ABB RobotStudio station: Mark3.rspag

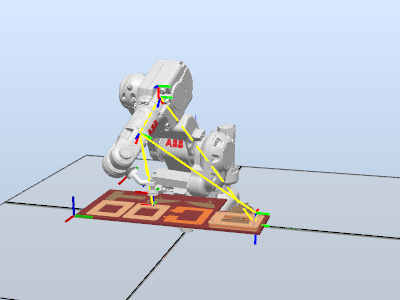
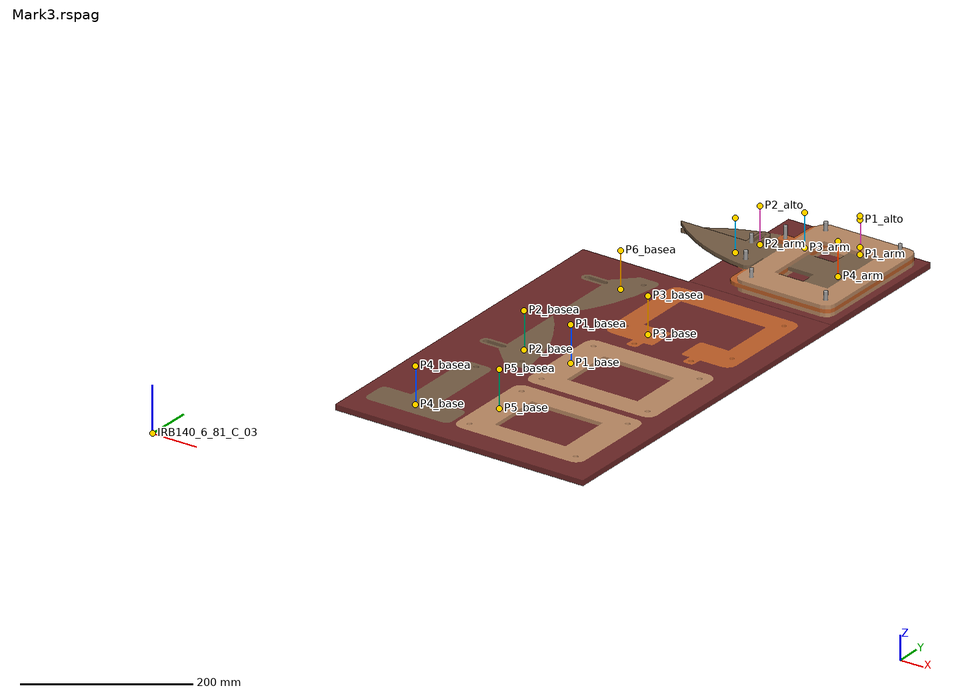
[picture v1: parts stored in the station drawn from their meshes, with robot base, taught points and paths (robot models come from the ABB library and are not in the file)]
--- station ---
Station Mark2 (saved by RobotStudio 22.2.9947.0)
Controller ControladorProyecto
  mechanical unit ROB_1: IRB140_6_81_C_03, 6 joints, base frame (0, 0, 0) mm
Layout (positions relative to the parent item):
  - IRB140_6_81_C_03 [mechanism, from Robots\IRB140_6_81_C_G_03.rslib] at (0, 0, 0) mm; joint values [-0.2236, 0.6546, -0.0796, 0.7946, 1.3157, -2.1338] (rad or m)
  - PortaPiezas [part] at (600, 0, 250) mm, rotated rx 0 ry 0 rz -90 deg, size 500 x 350 x 7 mm
  - BaseEnsamble [part] at (677, 353, 250) mm, rotated rx 0 ry 0 rz 180 deg, size 282.5 x 200 x 35 mm
  - Ventosa_AJDJ [mechanism] at (592.94, -88.78, 385.01) mm, rotated rx 180 ry 45.08 rz -90 deg
      TCP Ventosa_AJDJ at (-6, 0, 116) mm, rotated rx 0 ry 45 rz 0 deg
      links: portaherramienta
Attachment: Ventosa_AJDJ is attached to IRB140_6_81_C_03 / Link6

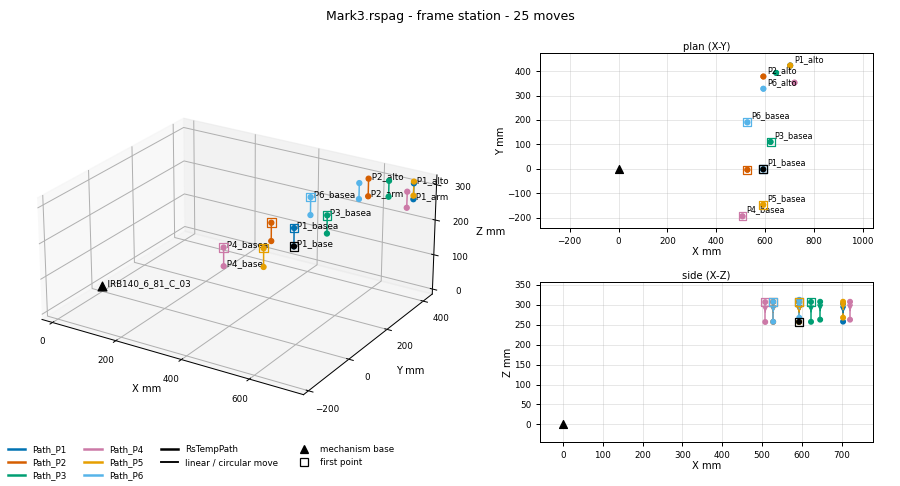
[picture p0: tool path of Mark3.rspag in frame station, 25 of 51 moves have a stored position in this frame; points joined in program order, loops and branches not executed]
--- Backups/ControladorProyecto/RAPID/TASK1/PROGMOD/CalibData.mod ---
MODULE CalibData
    PERS tooldata Ventosa_AJDJ:=[TRUE,[[-6,0,116],[0.923879533,0,0.382683432,0]],[0.15,[0,0,1],[1,0,0,0],0,0,0]];
    TASK PERS wobjdata Objeto_AJDJ:=[FALSE,TRUE,"",[[780.94,-246.929,257],[0.999999745,0.000714088,0,0]],[[0,0,0],[1,0,0,0]]];
ENDMODULE

--- Backups/ControladorProyecto/RAPID/TASK1/PROGMOD/Module1.mod ---
MODULE Module1
    CONST jointtarget Home:=[[0,0,0,0,45,0],[9E+09,9E+09,9E+09,9E+09,9E+09,9E+09]];
    CONST jointtarget P1_aux:=[[-5,20,0,-50,-10,25],[9E+09,9E+09,9E+09,9E+09,9E+09,9E+09]];
    CONST robtarget P1_basea:=[[-188,244.6,50],[0,-0.707106781,0.707106781,0],[-1,0,-2,0],[9E+09,9E+09,9E+09,9E+09,9E+09,9E+09]];
    CONST robtarget P1_base:=[[-188,244.6,0],[0,-0.707106781,0.707106781,0],[-1,0,-2,0],[9E+09,9E+09,9E+09,9E+09,9E+09,9E+09]];
    CONST robtarget P1_alto:=[[-77.5,670,45],[0,0,1,0],[0,1,-2,1],[9E+09,9E+09,9E+09,9E+09,9E+09,9E+09]];
    CONST robtarget P1_arm:=[[-77.5,670,0],[0,0,1,0],[0,1,-2,1],[9E+09,9E+09,9E+09,9E+09,9E+09,9E+09]];
    CONST jointtarget P2_aux:=[[0,20,20,-2,-5,0],[9E+09,9E+09,9E+09,9E+09,9E+09,9E+09]];
    CONST robtarget P2_basea:=[[-253,242.9,50],[0,0,1,0],[-1,-1,0,1],[9E+09,9E+09,9E+09,9E+09,9E+09,9E+09]];
    CONST robtarget P2_base:=[[-253,242.9,0],[0,0,1,0],[-1,-1,0,1],[9E+09,9E+09,9E+09,9E+09,9E+09,9E+09]];
    CONST robtarget P2_alto:=[[-187.5,625,50],[0,-0.707106781,0.707106781,0],[0,-2,0,1],[9E+09,9E+09,9E+09,9E+09,9E+09,9E+09]];
    CONST robtarget P2_arm:=[[-187.5,625,0],[0,-0.707106781,0.707106781,0],[0,-2,0,1],[9E+09,9E+09,9E+09,9E+09,9E+09,9E+09]];
    CONST jointtarget P3_aux:=[[0,20,-5,25,25,-40],[9E+09,9E+09,9E+09,9E+09,9E+09,9E+09]];
    CONST robtarget P3_basea:=[[-158,357.12,50],[0,-0.707106781,0.707106781,0],[-1,0,-2,0],[9E+09,9E+09,9E+09,9E+09,9E+09,9E+09]];
    CONST robtarget P3_base:=[[-158,357.12,0],[0,-0.707106781,0.707106781,0],[-1,0,-2,0],[9E+09,9E+09,9E+09,9E+09,9E+09,9E+09]];
    CONST robtarget P3_alto:=[[-135,640,50],[0,0,1,0],[0,-1,0,0],[9E+09,9E+09,9E+09,9E+09,9E+09,9E+09]];
    CONST robtarget P3_arm:=[[-135,640,5],[0,0,1,0],[0,-1,0,0],[9E+09,9E+09,9E+09,9E+09,9E+09,9E+09]];
    CONST jointtarget P4_aux:=[[-10,10,10,50,10,-50],[9E+09,9E+09,9E+09,9E+09,9E+09,9E+09]];
    CONST robtarget P4_basea:=[[-273,52.1,50],[0,0,1,0],[-1,0,-2,0],[9E+09,9E+09,9E+09,9E+09,9E+09,9E+09]];
    CONST robtarget P4_base:=[[-273,52.1,0],[0,0,1,0],[-1,1,-2,0],[9E+09,9E+09,9E+09,9E+09,9E+09,9E+09]];
    CONST robtarget P4_alto:=[[-60,600,50],[0,-0.707106781,0.707106781,0],[0,0,-1,0],[9E+09,9E+09,9E+09,9E+09,9E+09,9E+09]];
    CONST robtarget P4_arm:=[[-60,600,5],[0,-0.707106781,0.707106781,0],[0,0,-2,0],[9E+09,9E+09,9E+09,9E+09,9E+09,9E+09]];
    CONST jointtarget P5_aux:=[[-15,20,-5,20,50,-50],[9E+09,9E+09,9E+09,9E+09,9E+09,9E+09]];
    CONST robtarget P5_basea:=[[-188,99.7,50],[0,-0.707106781,0.707106781,0],[-1,0,-2,0],[9E+09,9E+09,9E+09,9E+09,9E+09,9E+09]];
    CONST robtarget P5_base:=[[-188,99.7,0],[0,-0.707106781,0.707106781,0],[-1,0,-2,0],[9E+09,9E+09,9E+09,9E+09,9E+09,9E+09]];
    CONST robtarget P5_alto:=[[-77.5,670,50],[0,0,1,0],[0,-1,0,0],[9E+09,9E+09,9E+09,9E+09,9E+09,9E+09]];
    CONST robtarget P5_arm:=[[-77.5,670,10],[0,0,1,0],[0,-1,0,0],[9E+09,9E+09,9E+09,9E+09,9E+09,9E+09]];
    CONST jointtarget P6_aux:=[[10,10,10,-50,5,50],[9E+09,9E+09,9E+09,9E+09,9E+09,9E+09]];
    CONST robtarget P6_basea:=[[-253,437.2,50],[0,0,1,0],[0,-1,1,0],[9E+09,9E+09,9E+09,9E+09,9E+09,9E+09]];
    CONST robtarget P6_base:=[[-253,437.2,0],[0,0,1,0],[0,-2,1,0],[9E+09,9E+09,9E+09,9E+09,9E+09,9E+09]];
    CONST robtarget P6_alto:=[[-187.5,575,55],[0,0.707106781,0.707106781,0],[0,-1,1,0],[9E+09,9E+09,9E+09,9E+09,9E+09,9E+09]];
    CONST robtarget P6_arm:=[[-187.5,575,10],[0,0.707106781,0.707106781,0],[0,-1,1,0],[9E+09,9E+09,9E+09,9E+09,9E+09,9E+09]];
    CONST jointtarget Home_lab:=[[0,0,0,0,0,0],[9E+09,9E+09,9E+09,9E+09,9E+09,9E+09]];
    PROC Path_P1()
        MoveAbsJ Home,v100,z10,Ventosa_AJDJ\WObj:=Objeto_AJDJ;
        MoveAbsJ P1_aux,v100,z10,Ventosa_AJDJ\WObj:=Objeto_AJDJ;
        MoveL P1_basea,v50,z10,Ventosa_AJDJ\WObj:=Objeto_AJDJ;
        MoveL P1_base,v100,z10,Ventosa_AJDJ\WObj:=Objeto_AJDJ;
        WaitDI DI_01,1;
        SetDO DO_01,1;
        SetDO DO_01,0;
        MoveAbsJ P1_aux,v100,z10,Ventosa_AJDJ\WObj:=Objeto_AJDJ;
        MoveL P1_alto,v100,z10,Ventosa_AJDJ\WObj:=Objeto_AJDJ;
        MoveL P1_arm,v100,z10,Ventosa_AJDJ\WObj:=Objeto_AJDJ;
        WaitDI DI_01,1;
        SetDO DO_02,1;
        SetDO DO_02,0;
        MoveAbsJ Home,v100,z10,Ventosa_AJDJ\WObj:=Objeto_AJDJ;
    ENDPROC
    PROC Path_P2()
        MoveAbsJ Home,v100,z10,Ventosa_AJDJ\WObj:=Objeto_AJDJ;
        MoveAbsJ P2_aux,v100,z10,Ventosa_AJDJ\WObj:=Objeto_AJDJ;
        MoveL P2_basea,v50,z10,Ventosa_AJDJ\WObj:=Objeto_AJDJ;
        MoveL P2_base,v100,z10,Ventosa_AJDJ\WObj:=Objeto_AJDJ;
        WaitDI DI_01,1;
        SetDO DO_01,1;
        SetDO DO_01,0;
        MoveAbsJ P2_aux,v100,z10,Ventosa_AJDJ\WObj:=Objeto_AJDJ;
        MoveL P2_alto,v100,z10,Ventosa_AJDJ\WObj:=Objeto_AJDJ;
        MoveL P2_arm,v100,z10,Ventosa_AJDJ\WObj:=Objeto_AJDJ;
        WaitDI DI_01,1;
        SetDO DO_02,1;
        SetDO DO_02,0;
        MoveAbsJ Home,v100,z10,Ventosa_AJDJ\WObj:=Objeto_AJDJ;
    ENDPROC
    PROC Path_P3()
        MoveAbsJ Home,v100,z10,Ventosa_AJDJ\WObj:=Objeto_AJDJ;
        MoveAbsJ P3_aux,v100,z10,Ventosa_AJDJ\WObj:=Objeto_AJDJ;
        MoveL P3_basea,v50,z10,Ventosa_AJDJ\WObj:=Objeto_AJDJ;
        MoveL P3_base,v100,z10,Ventosa_AJDJ\WObj:=Objeto_AJDJ;
        WaitDI DI_01,1;
        SetDO DO_01,1;
        SetDO DO_01,0;
        MoveAbsJ P3_aux,v100,z10,Ventosa_AJDJ\WObj:=Objeto_AJDJ;
        MoveL P3_alto,v100,z10,Ventosa_AJDJ\WObj:=Objeto_AJDJ;
        MoveL P3_arm,v100,z10,Ventosa_AJDJ\WObj:=Objeto_AJDJ;
        WaitDI DI_01,1;
        SetDO DO_02,1;
        SetDO DO_02,0;
        MoveAbsJ Home,v100,z10,Ventosa_AJDJ\WObj:=Objeto_AJDJ;
    ENDPROC
    PROC Path_P4()
        MoveAbsJ Home,v100,z10,Ventosa_AJDJ\WObj:=Objeto_AJDJ;
        MoveAbsJ P4_aux,v100,z10,Ventosa_AJDJ\WObj:=Objeto_AJDJ;
        MoveL P4_basea,v50,z10,Ventosa_AJDJ\WObj:=Objeto_AJDJ;
        MoveL P4_base,v100,z10,Ventosa_AJDJ\WObj:=Objeto_AJDJ;
        WaitDI DI_01,1;
        SetDO DO_01,1;
        SetDO DO_01,0;
        MoveAbsJ P4_aux,v100,z10,Ventosa_AJDJ\WObj:=Objeto_AJDJ;
        MoveL P4_alto,v100,z10,Ventosa_AJDJ\WObj:=Objeto_AJDJ;
        MoveL P4_arm,v100,z10,Ventosa_AJDJ\WObj:=Objeto_AJDJ;
        WaitDI DI_01,1;
        SetDO DO_02,1;
        SetDO DO_02,0;
        MoveAbsJ Home,v100,z10,Ventosa_AJDJ\WObj:=Objeto_AJDJ;
    ENDPROC
    PROC Path_P5()
        MoveAbsJ Home,v100,z10,Ventosa_AJDJ\WObj:=Objeto_AJDJ;
        MoveAbsJ P5_aux,v100,z10,Ventosa_AJDJ\WObj:=Objeto_AJDJ;
        MoveL P5_basea,v50,z10,Ventosa_AJDJ\WObj:=Objeto_AJDJ;
        MoveL P5_base,v100,z10,Ventosa_AJDJ\WObj:=Objeto_AJDJ;
        WaitDI DI_01,1;
        SetDO DO_01,1;
        SetDO DO_01,0;
        MoveAbsJ P5_aux,v100,z10,Ventosa_AJDJ\WObj:=Objeto_AJDJ;
        MoveL P5_alto,v100,z10,Ventosa_AJDJ\WObj:=Objeto_AJDJ;
        MoveL P5_arm,v100,z10,Ventosa_AJDJ\WObj:=Objeto_AJDJ;
        WaitDI DI_01,1;
        SetDO DO_02,1;
        SetDO DO_02,0;
        MoveAbsJ Home,v100,z10,Ventosa_AJDJ\WObj:=Objeto_AJDJ;
        MoveAbsJ P5_aux,v100,z10,Ventosa_AJDJ\WObj:=Objeto_AJDJ;
    ENDPROC
    PROC Path_P6()
        MoveAbsJ Home,v100,z10,Ventosa_AJDJ\WObj:=Objeto_AJDJ;
        MoveAbsJ P6_aux,v100,z10,Ventosa_AJDJ\WObj:=Objeto_AJDJ;
        MoveL P6_basea,v50,z10,Ventosa_AJDJ\WObj:=Objeto_AJDJ;
        MoveL P6_base,v100,z10,Ventosa_AJDJ\WObj:=Objeto_AJDJ;
        WaitDI DI_01,1;
        SetDO DO_01,1;
        SetDO DO_01,0;
        MoveAbsJ P6_aux,v100,z10,Ventosa_AJDJ\WObj:=Objeto_AJDJ;
        MoveL P6_alto,v100,z10,Ventosa_AJDJ\WObj:=Objeto_AJDJ;
        MoveL P6_arm,v100,z10,Ventosa_AJDJ\WObj:=Objeto_AJDJ;
        WaitDI DI_01,1;
        SetDO DO_02,1;
        SetDO DO_02,0;
        MoveAbsJ Home,v100,z10,Ventosa_AJDJ\WObj:=Objeto_AJDJ;
    ENDPROC
    PROC main()
        WaitDI DI_01,1;
        ToHome;
        WaitDI DI_01,1;
        Path_P1;
        Path_P2;
        Path_P3;
        Path_P4;
        Path_P5;
        Path_P6;
        ToHome;
        SetDO DO_01,1;
    ENDPROC
    PROC ToHome()
        MoveAbsJ Home_lab,v1000,z100,Ventosa_AJDJ\WObj:=Objeto_AJDJ;
    ENDPROC
ENDMODULE

--- Backups/ControladorProyecto/RAPID/TASK1/PROGMOD/RsTempModule.mod ---
MODULE RsTempModule
    LOCAL CONST robtarget P1_base:=[[-188,244.6,0],[0,-0.707106781,0.707106781,0],[-1,0,-2,0],[9E+09,9E+09,9E+09,9E+09,9E+09,9E+09]];
    LOCAL PERS tooldata Ventosa_AJDJ:=[TRUE,[[-6,0,116],[0.923879533,0,0.382683432,0]],[0.15,[0,0,1],[1,0,0,0],0,0,0]];
    LOCAL PERS wobjdata Objeto_AJDJ:=[FALSE,TRUE,"",[[780.94,-246.929,257],[0.999999745,0.000714088,0,0]],[[0,0,0],[1,0,0,0]]];
PROC RsTempPath()
        MoveL P1_base,v100,z10,Ventosa_AJDJ\WObj:=Objeto_AJDJ;
ENDPROC

ENDMODULE

--- Backups/ControladorProyecto/SYSPAR/EIO.cfg ---
EIO:CFG_1.0:6:1::
#
EIO_SIGNAL:

      -Name "DO_01" -SignalType "DO"

      -Name "DI_01" -SignalType "DI"

      -Name "DO_02" -SignalType "DO"
